FUNCTION_BLOCK FB_HartingIO

VAR_IN_OUT CONSTANT
	st_params 			: ST_HartingIO_params;
END_VAR

VAR_INPUT
	set 				: ST_HartingIO_Set;
	SystemOperating		: BOOL;
	SystemEmStop		: BOOL;
END_VAR

VAR_OUTPUT
	Get								:	ST_HartingIO_Get;
	b_SystemRestartTrigger			: 	BOOL;
END_VAR

VAR	
	b_ExtDO1				AT %Q* : BOOL;	
	b_ExtDO2				AT %Q* : BOOL;
	b_ExtDI1				AT %I* : BOOL;
	b_ExtDI2				AT %I* : BOOL;
	i_AO1					AT %Q* : INT;
	i_AO2					AT %Q* : INT;
END_VAR

b_ExtDO1 := configureOutputContact(SignalSelect := st_params.PrimaryOutputContactSignal); 
b_ExtDO2 := configureOutputContact(SignalSelect := st_params.SecondaryOutputContactSignal); 
 
configureInputcontact(SignalSelect := st_params.PrimaryInputContactSignal, b_ExtDI1); 
//configureInputcontact(SignalSelect := st_params.SecondaryInputContactSignal, b_ExtDI2); 
get.b_DigitalInput1Active := b_ExtDi1;
get.b_DigitalInput2Active := b_ExtDi2;

AutoRestartAfterExtEmstop();


CASE st_params.AO1Target OF
	eAOtarget.manual	: i_AO1 := AnalogOutputScaling(set.r_manualAnalogOutput);
	eAOtarget.Genset	: i_AO1 := AnalogOutputScaling(set.r_gensetAnalogOutput);
	eAOtarget.hPU		: i_AO1 := AnalogOutputScaling(set.r_HpuAnalogOutput);
END_CASE

CASE st_params.AO2Target OF
	eAOtarget.manual	: i_AO2 := AnalogOutputScaling(set.r_manualAnalogOutput);
	eAOtarget.Genset	: i_AO2 := AnalogOutputScaling(set.r_gensetAnalogOutput);
	eAOtarget.hPU		: i_AO2 := AnalogOutputScaling(set.r_HpuAnalogOutput);
END_CASE

METHOD AnalogOutputScaling : INT
VAR_INPUT
	IN : REAL;
END_VAR

VAR_INST
	scale_analogOutput			: FB_ctrl_Scale;
	st_paramsScale				: ST_ctrl_scale_params;
END_VAR
//Scale real to analog output
st_paramsScale.fInMax:= 100;
	st_paramsScale.fInMin:= 0;
	st_paramsScale.fOutMax:= 16#8000 -1;
	st_paramsScale.fOutMin:= 0;
	st_paramsScale.tCtrlCycleTime := T#1MS;
	st_paramsScale.tTaskCycleTime := T#1MS;

scale_analogOutput(stParams:= st_paramsScale,
	fIn:= IN);
	AnalogOutputScaling := TO_INT(scale_analogOutput.fOut);
END_METHOD

METHOD AutoRestartAfterExtEmstop : BOOL
VAR_INST
	SystemLastOperation : BOOL;
	
	ExtEmStopRestartTriggered	: BOOL;
	R_TrigoperatingReset		: R_TRIG;
	Ton_DelayCheckState	: TON := (PT:=T#2S);	
END_VAR
IF get.b_ExtEMstopActive THEN
	ExtEmStopRestartTriggered := TRUE;
END_IF

R_TrigoperatingReset(CLK := SystemOperating);
IF R_TrigoperatingReset.Q AND ExtEmStopRestartTriggered THEN
	ExtEmStopRestartTriggered := FALSE;
END_IF

IF NOT SystemEmStop AND SystemOperating THEN
	SystemLastOperation := TRUE;
END_IF

Ton_DelayCheckState(IN := NOT ExtEmStopRestartTriggered AND NOT SystemOperating);
IF ton_DelayCheckState.Q THEN
	SystemLastOperation := FALSE;
END_IF

b_SystemRestartTrigger := SystemLastOperation AND ExtEmStopRestartTriggered;
END_METHOD

METHOD ConfigureInputContact : BOOL
VAR_INPUT
	SignalSelect			: 	eInputSignal;
	InputStatus				:	BOOL;
END_VAR
get.b_GenLowFuel 				:= (SignalSelect = eInputSignal.GenLowFuel) 	AND InputStatus;
get.b_ExtSystemShutdownRequest 	:= (SignalSelect = eInputSignal.StopOperation) 	AND InputStatus;
get.b_ExtEmstopOK 				:= (SignalSelect = eInputSignal.EMstop) 		AND InputStatus;
END_METHOD

METHOD ConfigureOutputContact : BOOL
VAR_INPUT
	SignalSelect			: eOutputContactSignal;
END_VAR
CASE SignalSelect OF
	eOutputContactSignal.GenStartStop 	: ConfigureOutputContact:= set.w_SwitchControlSignals.0;
	eOutputContactSignal.FireAlarm 		: ConfigureOutputContact:= set.w_SwitchControlSignals.1;
	eOutputContactSignal.HPU			: ConfigureOutputContact:= set.w_SwitchControlSignals.2;
	eOutputContactSignal.SystemActive	: ConfigureOutputContact:= set.w_SwitchControlSignals.3;
	eOutputContactSignal.PVenable		: ConfigureOutputContact:= set.w_SwitchControlSignals.4;
	eOutputContactSignal.None, eOutputContactSignal.ManualOpen	
										:	ConfigureOutputContact := FALSE;
	eOutputContactSignal.ManualClose	:	ConfigureOutputContact := TRUE;
END_CASE
END_METHOD

METHOD GetDiagnostics
VAR_IN_OUT
	AddError		: ARRAY [*] OF FB_AddErrorST;
	a_ActiveEvents	: ARRAY [*] OF ST_ErrorStruct;
	w_Index			: WORD;
END_VAR
	(*Shutdown trigger*)		AddError[w_Index](
					b_ErrorTrig				:= get.b_ExtSystemShutdownRequest,
					out_ST_Error			:= a_ActiveEvents[w_Index],
					w_ErrorID				:= 1,
					e_ObjectID				:= eObject_ID.HartingIO,
					s_Message				:= 'External shutdown triggered',
					e_sev					:= eSeverity.NormalShutdown
				);
				w_Index := w_Index +1;
				
		(*EMstop trigger*)		AddError[w_Index](
					b_ErrorTrig				:= ((st_params.PrimaryInputContactSignal = eInputSignal.emstop) OR (st_params.SecondaryInputContactSignal = eInputSignal.emstop)) AND NOT get.b_ExtEMstopOK,
					out_ST_Error			:= a_ActiveEvents[w_Index],
					w_ErrorID				:= 2,
					e_ObjectID				:= eObject_ID.HartingIO,
					s_Message				:= 'External EMstop triggered',
					e_sev					:= eSeverity.QuickShutdown,
					b_Out					=> get.b_ExtEMstopActive
				);
				w_Index := w_Index +1;
END_METHOD

END_FUNCTION_BLOCK

(* stored: Version 1.1.0.1, ProductVersion 3.1.4026.18
   POU FB_HartingIO: Id {a67e4543-1657-497c-847b-a125d1a62217}, SpecialFunc None
   Method AnalogOutputScaling: Id {a93d90e8-d581-4009-ba4f-2142021827bc}
   Method AutoRestartAfterExtEmstop: Id {5258782f-e64f-42a8-a3ff-73f3c8271db9}
   Method ConfigureInputContact: Id {b9ea5b96-dc66-4583-8ae9-acc3e46496c4}
   Method ConfigureOutputContact: Id {4099e2c1-f345-4088-9f53-d0e1b8c3d15c}
   Method GetDiagnostics: Id {09b3e139-dadc-4a0f-b8dd-64b7d9504b4b} *)
